Yaskawa INFORM job: u_profile_planes_program.JBI

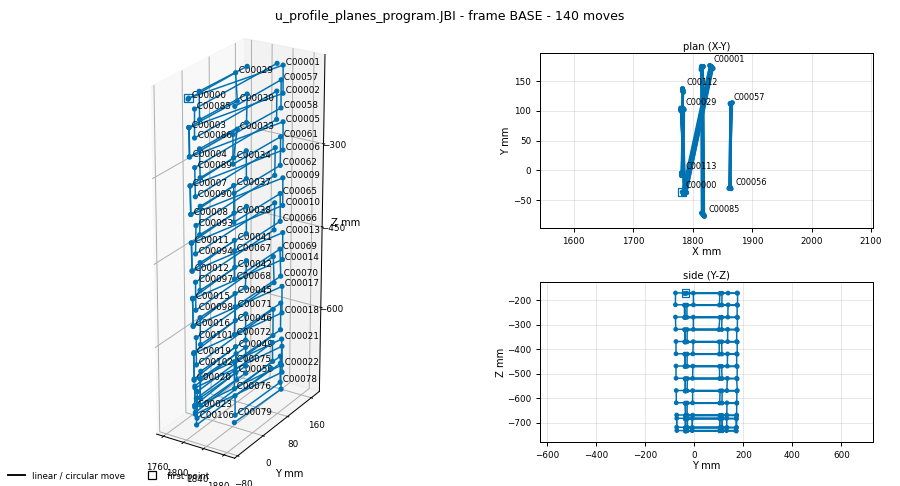
[picture p0: tool path of u_profile_planes_program.JBI in frame BASE, 140 of 146 moves have a stored position in this frame; points joined in program order, loops and branches not executed]
/JOB
//NAME u_profile_planes_program
//POS
///NPOS 140,0,140,0,0,0
///TOOL 0
///POSTYPE BASE
///RECTAN
///RCONF 0,0,0,0,0,0,0,0,0,0,0,0,0,0,0,0,0,0,0,0,0,0,0,0
C00000=1782.260933,-36.525001,-172.991933,5.000000,-89.396315,175.000000
C00001=1828.522430,176.080910,-172.464525,5.000000,-89.396315,175.000000
C00002=1828.739389,176.154104,-221.512851,5.000000,-89.396315,175.000000
C00003=1783.694118,-38.162419,-222.027765,5.000000,-89.396315,175.000000
C00004=1783.978818,-37.816790,-272.027476,5.000000,-89.396315,175.000000
C00005=1829.604124,175.680714,-271.506605,5.000000,-89.396315,175.000000
C00006=1830.194434,175.105438,-321.503269,5.000000,-89.396315,175.000000
C00007=1784.623679,-37.894376,-322.023473,5.000000,-89.396315,175.000000
C00008=1784.583709,-36.947245,-372.026492,5.000000,-89.396315,175.000000
C00009=1830.568449,174.887024,-371.502146,5.000000,-89.396315,175.000000
C00010=1830.901280,174.569844,-421.501475,5.000000,-89.396315,175.000000
C00011=1786.103914,-37.913551,-422.013432,5.000000,-89.396315,175.000000
C00012=1786.618585,-37.695016,-472.010744,5.000000,-89.396315,175.000000
C00013=1831.454807,174.703887,-471.498394,5.000000,-89.396315,175.000000
C00014=1831.389630,174.529477,-521.501890,5.000000,-89.396315,175.000000
C00015=1786.911299,-37.647433,-522.010428,5.000000,-89.396315,175.000000
C00016=1787.341155,-37.497572,-572.008647,5.000000,-89.396315,175.000000
C00017=1831.659589,173.248889,-571.502062,5.000000,-89.396315,175.000000
C00018=1832.203103,172.929218,-621.499172,5.000000,-89.396315,175.000000
C00019=1787.872410,-37.676480,-622.005859,5.000000,-89.396315,175.000000
C00020=1787.809102,-36.881874,-672.009153,5.000000,-89.396315,175.000000
C00021=1832.658785,172.057548,-671.497311,5.000000,-89.396315,175.000000
C00022=1833.373411,171.254768,-721.492708,5.000000,-89.396315,175.000000
C00023=1789.315318,-37.854407,-721.996241,5.000000,-89.396315,175.000000
C00024=1789.930204,-37.686084,-685.389967,5.000000,-89.396315,175.000000
C00025=1833.724582,171.553342,-684.889188,5.000000,-89.396315,175.000000
C00026=1834.546973,171.110071,-734.883382,5.000000,-89.396315,175.000000
C00027=1790.024475,-37.371069,-735.391691,180.000000,-60.000000,0.000000
C00028=1784.263677,-41.032279,-172.869038,5.000000,-89.672423,175.000000
C00029=1781.616383,104.028574,-172.862041,5.000000,-89.672423,175.000000
C00030=1786.087872,101.937924,-220.615691,5.000000,-89.672423,175.000000
C00031=1784.435636,-40.713206,-220.646900,5.000000,-89.672423,175.000000
C00032=1784.974466,-40.445319,-270.644596,5.000000,-89.672423,175.000000
C00033=1784.613661,104.150813,-270.624599,5.000000,-89.672423,175.000000
C00034=1780.229983,99.510054,-320.651186,5.000000,-89.672423,175.000000
C00035=1785.412002,-40.051621,-320.642853,5.000000,-89.672423,175.000000
C00036=1785.985604,-39.459139,-370.640301,5.000000,-89.672423,175.000000
C00037=1779.523904,101.128963,-370.655793,5.000000,-89.672423,175.000000
C00038=1779.816005,101.531303,-420.654880,5.000000,-89.672423,175.000000
C00039=1786.350977,-39.228229,-420.638994,5.000000,-89.672423,175.000000
C00040=1786.742769,-38.468907,-470.637456,5.000000,-89.672423,175.000000
C00041=1780.262080,102.230709,-470.653041,5.000000,-89.672423,175.000000
C00042=1780.395302,102.757357,-520.653016,5.000000,-89.672423,175.000000
C00043=1786.735924,-37.738008,-520.638202,5.000000,-89.672423,175.000000
C00044=1787.164139,-37.411963,-570.636521,5.000000,-89.672423,175.000000
C00045=1779.566447,104.826652,-570.658257,5.000000,-89.672423,175.000000
C00046=1781.202178,103.217633,-620.649968,5.000000,-89.672423,175.000000
C00047=1787.638777,-36.535127,-620.634492,5.000000,-89.672423,175.000000
C00048=1786.878712,-35.395784,-670.639481,5.000000,-89.672423,175.000000
C00049=1781.436614,103.551324,-670.649395,5.000000,-89.672423,175.000000
C00050=1781.577028,104.048799,-720.649334,5.000000,-89.672423,175.000000
C00051=1787.065054,-34.835771,-720.639148,5.000000,-89.672423,175.000000
C00052=1787.558849,-34.268309,-684.034515,5.000000,-89.672423,175.000000
C00053=1782.466992,103.465471,-684.042612,5.000000,-89.672423,175.000000
C00054=1783.620917,103.201260,-734.036873,5.000000,-89.672423,175.000000
C00055=1787.804559,-33.884165,-734.033870,180.000000,-60.000000,0.000000
C00056=1864.910662,-31.222999,-172.174385,5.000000,-89.728805,175.000000
C00057=1863.073927,112.319586,-172.126552,5.000000,-89.728805,175.000000
C00058=1863.206204,112.281534,-220.384319,5.000000,-89.728805,175.000000
C00059=1860.927322,-30.501787,-220.451331,5.000000,-89.728805,175.000000
C00060=1861.061629,-30.477059,-270.451249,5.000000,-89.728805,175.000000
C00061=1862.988161,112.262490,-270.385923,5.000000,-89.728805,175.000000
C00062=1863.111960,111.513040,-320.386196,5.000000,-89.728805,175.000000
C00063=1862.283204,-29.603927,-320.445688,5.000000,-89.728805,175.000000
C00064=1861.955339,-29.823655,-370.447890,5.000000,-89.728805,175.000000
C00065=1863.459829,111.554401,-370.385097,5.000000,-89.728805,175.000000
C00066=1863.578969,111.994231,-420.384924,5.000000,-89.728805,175.000000
C00067=1862.661633,-29.633452,-420.445036,5.000000,-89.728805,175.000000
C00068=1862.840974,-29.862305,-470.444841,5.000000,-89.728805,175.000000
C00069=1864.119807,111.277161,-470.383210,5.000000,-89.728805,175.000000
C00070=1865.056679,112.773774,-520.378751,5.000000,-89.728805,175.000000
C00071=1863.450288,-28.702334,-520.442065,5.000000,-89.728805,175.000000
C00072=1862.667533,-29.829051,-570.446777,5.000000,-89.728805,175.000000
C00073=1865.408367,113.053169,-570.377540,5.000000,-89.728805,175.000000
C00074=1865.447046,112.860239,-620.377997,5.000000,-89.728805,175.000000
C00075=1862.411067,-29.646174,-620.448483,5.000000,-89.728805,175.000000
C00076=1862.548753,-29.578278,-670.448368,5.000000,-89.728805,175.000000
C00077=1865.658542,112.889085,-670.377548,5.000000,-89.728805,175.000000
C00078=1865.699326,112.725750,-720.377983,5.000000,-89.728805,175.000000
C00079=1863.047601,-28.320485,-720.446076,5.000000,-89.728805,175.000000
C00080=1863.141010,-28.432178,-683.843701,5.000000,-89.728805,175.000000
C00081=1866.035142,112.824822,-683.774379,5.000000,-89.728805,175.000000
C00082=1866.942476,113.818457,-733.770257,5.000000,-89.728805,175.000000
C00083=1862.456330,-29.699196,-733.848004,180.000000,-60.000000,0.000000
C00084=1817.720355,174.738669,-171.016448,175.000000,-89.849838,5.000000
C00085=1819.771577,-77.235879,-171.008002,175.000000,-89.849838,5.000000
C00086=1819.536110,-77.464714,-219.320565,175.000000,-89.849838,5.000000
C00087=1817.731724,174.427635,-219.329654,175.000000,-89.849838,5.000000
C00088=1817.734630,174.455568,-269.329835,175.000000,-89.849838,5.000000
C00089=1819.232730,-77.296831,-269.319951,175.000000,-89.849838,5.000000
C00090=1819.307321,-76.203642,-319.320379,175.000000,-89.849838,5.000000
C00091=1816.598926,172.687935,-319.326933,175.000000,-89.849838,5.000000
C00092=1816.003565,172.546900,-369.325537,175.000000,-89.849838,5.000000
C00093=1819.307141,-75.128762,-369.320609,175.000000,-89.849838,5.000000
C00094=1817.949037,-75.148117,-419.317220,175.000000,-89.849838,5.000000
C00095=1816.368409,172.540616,-419.326665,175.000000,-89.849838,5.000000
C00096=1815.455446,172.524070,-469.324443,175.000000,-89.849838,5.000000
C00097=1817.440701,-75.186175,-469.316057,175.000000,-89.849838,5.000000
C00098=1817.453052,-75.033079,-519.316270,175.000000,-89.849838,5.000000
C00099=1814.325290,172.534919,-519.321653,175.000000,-89.849838,5.000000
C00100=1814.693928,174.998074,-569.322926,175.000000,-89.849838,5.000000
C00101=1817.184370,-74.226679,-569.315782,175.000000,-89.849838,5.000000
C00102=1817.012743,-74.091457,-619.315511,175.000000,-89.849838,5.000000
C00103=1814.499495,172.911626,-619.322474,175.000000,-89.849838,5.000000
C00104=1814.813610,172.267579,-669.323434,175.000000,-89.849838,5.000000
C00105=1817.273302,-72.417306,-669.316458,175.000000,-89.849838,5.000000
C00106=1816.265495,-72.410539,-719.313989,175.000000,-89.849838,5.000000
C00107=1814.842076,171.681747,-719.323648,175.000000,-89.849838,5.000000
C00108=1814.465788,171.325455,-682.720274,175.000000,-89.849838,5.000000
C00109=1815.013489,-72.075161,-682.708357,175.000000,-89.849838,5.000000
C00110=1814.906208,-71.760453,-732.708265,175.000000,-89.849838,5.000000
C00111=1813.881604,169.060096,-732.718790,180.000000,-60.000000,0.000000
C00112=1782.888338,137.586668,-171.654258,5.000000,-89.861988,175.000000
C00113=1781.154819,-4.384120,-171.681020,5.000000,-89.861988,175.000000
C00114=1781.350773,-3.962780,-219.774254,5.000000,-89.861988,175.000000
C00115=1783.047830,137.404084,-219.747675,5.000000,-89.861988,175.000000
C00116=1782.612125,136.250340,-269.749054,5.000000,-89.861988,175.000000
C00117=1781.075396,-4.466191,-269.775143,5.000000,-89.861988,175.000000
C00118=1781.746415,-4.325570,-319.773650,5.000000,-89.861988,175.000000
C00119=1782.510065,135.829048,-319.749513,5.000000,-89.861988,175.000000
C00120=1782.978582,135.477793,-369.748586,5.000000,-89.861988,175.000000
C00121=1781.750223,-4.776320,-369.773858,5.000000,-89.861988,175.000000
C00122=1781.318160,-6.279225,-419.775283,5.000000,-89.861988,175.000000
C00123=1783.591949,135.128919,-419.747309,5.000000,-89.861988,175.000000
C00124=1783.512465,134.569931,-469.747735,5.000000,-89.861988,175.000000
C00125=1781.757069,-6.288375,-469.774373,5.000000,-89.861988,175.000000
C00126=1781.639717,-7.192765,-519.774946,5.000000,-89.861988,175.000000
C00127=1784.012555,134.399599,-519.746704,5.000000,-89.861988,175.000000
C00128=1782.981736,132.564435,-569.749624,5.000000,-89.861988,175.000000
C00129=1781.532036,-7.293985,-569.775367,5.000000,-89.861988,175.000000
C00130=1781.692072,-7.278391,-619.775124,5.000000,-89.861988,175.000000
C00131=1783.650110,132.855079,-619.748114,5.000000,-89.861988,175.000000
C00132=1783.771830,132.286276,-669.748057,5.000000,-89.861988,175.000000
C00133=1781.857171,-7.162989,-669.774854,5.000000,-89.861988,175.000000
C00134=1781.078721,-8.764395,-719.777130,5.000000,-89.861988,175.000000
C00135=1784.069920,132.313501,-719.747480,5.000000,-89.861988,175.000000
C00136=1784.401337,131.663006,-683.144391,5.000000,-89.861988,175.000000
C00137=1781.436060,-9.064609,-683.173922,5.000000,-89.861988,175.000000
C00138=1781.420701,-9.194187,-733.174125,5.000000,-89.861988,175.000000
C00139=1784.503273,131.243906,-733.144357,180.000000,-60.000000,0.000000
///POSTYPE PULSE
///PULSE
EC00000=2048.0
EC00001=2048.0
EC00002=2048.0
EC00003=2048.0
EC00004=2048.0
EC00005=2048.0
EC00006=2048.0
EC00007=2048.0
EC00008=2048.0
EC00009=2048.0
EC00010=2048.0
EC00011=2048.0
EC00012=2048.0
EC00013=2048.0
EC00014=2048.0
EC00015=2048.0
EC00016=2048.0
EC00017=2048.0
EC00018=2048.0
EC00019=2048.0
EC00020=2048.0
EC00021=2048.0
EC00022=2048.0
EC00023=2048.0
EC00024=2048.0
EC00025=2048.0
EC00026=2048.0
EC00027=2048.0
EC00028=95232.0
EC00029=95232.0
EC00030=95232.0
EC00031=95232.0
EC00032=95232.0
EC00033=95232.0
EC00034=95232.0
EC00035=95232.0
EC00036=95232.0
EC00037=95232.0
EC00038=95232.0
EC00039=95232.0
EC00040=95232.0
EC00041=95232.0
EC00042=95232.0
EC00043=95232.0
EC00044=95232.0
EC00045=95232.0
EC00046=95232.0
EC00047=95232.0
EC00048=95232.0
EC00049=95232.0
EC00050=95232.0
EC00051=95232.0
EC00052=95232.0
EC00053=95232.0
EC00054=95232.0
EC00055=95232.0
EC00056=102400.0
EC00057=102400.0
EC00058=102400.0
EC00059=102400.0
EC00060=102400.0
EC00061=102400.0
EC00062=102400.0
EC00063=102400.0
EC00064=102400.0
EC00065=102400.0
EC00066=102400.0
EC00067=102400.0
EC00068=102400.0
EC00069=102400.0
EC00070=102400.0
EC00071=102400.0
EC00072=102400.0
EC00073=102400.0
EC00074=102400.0
EC00075=102400.0
EC00076=102400.0
EC00077=102400.0
EC00078=102400.0
EC00079=102400.0
EC00080=102400.0
EC00081=102400.0
EC00082=102400.0
EC00083=102400.0
EC00084=186368.0
EC00085=186368.0
EC00086=186368.0
EC00087=186368.0
EC00088=186368.0
EC00089=186368.0
EC00090=186368.0
EC00091=186368.0
EC00092=186368.0
EC00093=186368.0
EC00094=186368.0
EC00095=186368.0
EC00096=186368.0
EC00097=186368.0
EC00098=186368.0
EC00099=186368.0
EC00100=186368.0
EC00101=186368.0
EC00102=186368.0
EC00103=186368.0
EC00104=186368.0
EC00105=186368.0
EC00106=186368.0
EC00107=186368.0
EC00108=186368.0
EC00109=186368.0
EC00110=186368.0
EC00111=186368.0
EC00112=284672.0
EC00113=284672.0
EC00114=284672.0
EC00115=284672.0
EC00116=284672.0
EC00117=284672.0
EC00118=284672.0
EC00119=284672.0
EC00120=284672.0
EC00121=284672.0
EC00122=284672.0
EC00123=284672.0
EC00124=284672.0
EC00125=284672.0
EC00126=284672.0
EC00127=284672.0
EC00128=284672.0
EC00129=284672.0
EC00130=284672.0
EC00131=284672.0
EC00132=284672.0
EC00133=284672.0
EC00134=284672.0
EC00135=284672.0
EC00136=284672.0
EC00137=284672.0
EC00138=284672.0
EC00139=284672.0
//INST
///DATE 2023/08/16 15:26
///ATTR SC,RW,RJ
////FRAME BASE
///GROUP1 RB1,ST1
NOP
MOVJ P009 EX000 VJ=15.00
MOVJ C00000 EC00000 VJ=15.0
CALL JOB:SPYON
MOVL C00001 EC00001 V=150.0
MOVL C00002 EC00002 V=150.0
MOVL C00003 EC00003 V=150.0
MOVL C00004 EC00004 V=150.0
MOVL C00005 EC00005 V=150.0
MOVL C00006 EC00006 V=150.0
MOVL C00007 EC00007 V=150.0
MOVL C00008 EC00008 V=150.0
MOVL C00009 EC00009 V=150.0
MOVL C00010 EC00010 V=150.0
MOVL C00011 EC00011 V=150.0
MOVL C00012 EC00012 V=150.0
MOVL C00013 EC00013 V=150.0
MOVL C00014 EC00014 V=150.0
MOVL C00015 EC00015 V=150.0
MOVL C00016 EC00016 V=150.0
MOVL C00017 EC00017 V=150.0
MOVL C00018 EC00018 V=150.0
MOVL C00019 EC00019 V=150.0
MOVL C00020 EC00020 V=150.0
MOVL C00021 EC00021 V=150.0
MOVL C00022 EC00022 V=150.0
MOVL C00023 EC00023 V=150.0
MOVL C00024 EC00024 V=150.0
MOVL C00025 EC00025 V=150.0
MOVL C00026 EC00026 V=150.0
MOVL C00027 EC00027 V=150.0
CALL JOB:SPYOF
MOVJ P009 VJ=15.00
MOVJ C00028 EC00028 VJ=15.0
CALL JOB:SPYON
MOVL C00029 EC00029 V=150.0
MOVL C00030 EC00030 V=150.0
MOVL C00031 EC00031 V=150.0
MOVL C00032 EC00032 V=150.0
MOVL C00033 EC00033 V=150.0
MOVL C00034 EC00034 V=150.0
MOVL C00035 EC00035 V=150.0
MOVL C00036 EC00036 V=150.0
MOVL C00037 EC00037 V=150.0
MOVL C00038 EC00038 V=150.0
MOVL C00039 EC00039 V=150.0
MOVL C00040 EC00040 V=150.0
MOVL C00041 EC00041 V=150.0
MOVL C00042 EC00042 V=150.0
MOVL C00043 EC00043 V=150.0
MOVL C00044 EC00044 V=150.0
MOVL C00045 EC00045 V=150.0
MOVL C00046 EC00046 V=150.0
MOVL C00047 EC00047 V=150.0
MOVL C00048 EC00048 V=150.0
MOVL C00049 EC00049 V=150.0
MOVL C00050 EC00050 V=150.0
MOVL C00051 EC00051 V=150.0
MOVL C00052 EC00052 V=150.0
MOVL C00053 EC00053 V=150.0
MOVL C00054 EC00054 V=150.0
MOVL C00055 EC00055 V=150.0
CALL JOB:SPYOF
MOVJ P009 VJ=15.00
MOVJ C00056 EC00056 VJ=15.0
CALL JOB:SPYON
MOVL C00057 EC00057 V=150.0
MOVL C00058 EC00058 V=150.0
MOVL C00059 EC00059 V=150.0
MOVL C00060 EC00060 V=150.0
MOVL C00061 EC00061 V=150.0
MOVL C00062 EC00062 V=150.0
MOVL C00063 EC00063 V=150.0
MOVL C00064 EC00064 V=150.0
MOVL C00065 EC00065 V=150.0
MOVL C00066 EC00066 V=150.0
MOVL C00067 EC00067 V=150.0
MOVL C00068 EC00068 V=150.0
MOVL C00069 EC00069 V=150.0
MOVL C00070 EC00070 V=150.0
MOVL C00071 EC00071 V=150.0
MOVL C00072 EC00072 V=150.0
MOVL C00073 EC00073 V=150.0
MOVL C00074 EC00074 V=150.0
MOVL C00075 EC00075 V=150.0
MOVL C00076 EC00076 V=150.0
MOVL C00077 EC00077 V=150.0
MOVL C00078 EC00078 V=150.0
MOVL C00079 EC00079 V=150.0
MOVL C00080 EC00080 V=150.0
MOVL C00081 EC00081 V=150.0
MOVL C00082 EC00082 V=150.0
MOVL C00083 EC00083 V=150.0
CALL JOB:SPYOF
MOVJ P009 VJ=15.00
MOVJ C00084 EC00084 VJ=15.0
CALL JOB:SPYON
MOVL C00085 EC00085 V=150.0
MOVL C00086 EC00086 V=150.0
MOVL C00087 EC00087 V=150.0
MOVL C00088 EC00088 V=150.0
MOVL C00089 EC00089 V=150.0
MOVL C00090 EC00090 V=150.0
MOVL C00091 EC00091 V=150.0
MOVL C00092 EC00092 V=150.0
MOVL C00093 EC00093 V=150.0
MOVL C00094 EC00094 V=150.0
MOVL C00095 EC00095 V=150.0
MOVL C00096 EC00096 V=150.0
MOVL C00097 EC00097 V=150.0
MOVL C00098 EC00098 V=150.0
MOVL C00099 EC00099 V=150.0
MOVL C00100 EC00100 V=150.0
MOVL C00101 EC00101 V=150.0
MOVL C00102 EC00102 V=150.0
MOVL C00103 EC00103 V=150.0
MOVL C00104 EC00104 V=150.0
MOVL C00105 EC00105 V=150.0
MOVL C00106 EC00106 V=150.0
MOVL C00107 EC00107 V=150.0
MOVL C00108 EC00108 V=150.0
MOVL C00109 EC00109 V=150.0
MOVL C00110 EC00110 V=150.0
MOVL C00111 EC00111 V=150.0
CALL JOB:SPYOF
MOVJ P009 VJ=15.00
MOVJ C00112 EC00112 VJ=15.0
CALL JOB:SPYON
MOVL C00113 EC00113 V=150.0
MOVL C00114 EC00114 V=150.0
MOVL C00115 EC00115 V=150.0
MOVL C00116 EC00116 V=150.0
MOVL C00117 EC00117 V=150.0
MOVL C00118 EC00118 V=150.0
MOVL C00119 EC00119 V=150.0
MOVL C00120 EC00120 V=150.0
MOVL C00121 EC00121 V=150.0
MOVL C00122 EC00122 V=150.0
MOVL C00123 EC00123 V=150.0
MOVL C00124 EC00124 V=150.0
MOVL C00125 EC00125 V=150.0
MOVL C00126 EC00126 V=150.0
MOVL C00127 EC00127 V=150.0
MOVL C00128 EC00128 V=150.0
MOVL C00129 EC00129 V=150.0
MOVL C00130 EC00130 V=150.0
MOVL C00131 EC00131 V=150.0
MOVL C00132 EC00132 V=150.0
MOVL C00133 EC00133 V=150.0
MOVL C00134 EC00134 V=150.0
MOVL C00135 EC00135 V=150.0
MOVL C00136 EC00136 V=150.0
MOVL C00137 EC00137 V=150.0
MOVL C00138 EC00138 V=150.0
MOVL C00139 EC00139 V=150.0
CALL JOB:SPYOF
MOVJ P009 VJ=15.00
END
